(*udt (user defined type) of Beckhoff EK1122 - EtherCAT Junction Terminal:
	auth. Brent Lekx-Toniolo of Toniolo Research & Development Inc.; 
	July 2010; version 1.0*)

TYPE udt_EK1122 :
STRUCT
	InfoData: udt_ECATSlave_Status;
END_STRUCT
END_TYPE

(* stored: Version 1.1.0.1, ProductVersion 3.1.4024.9
   DUT udt_EK1122: Id {44014dd9-589d-4b7b-ab65-a1c5aee7e7b7} *)
